TYPE DUT_DataRequest :
STRUCT
	aByte	: ARRAY[0..1] OF stByteAsBit; 	
	aDWord	: DWORD;
END_STRUCT
END_TYPE

(* stored: Version 1.1.0.1, ProductVersion 3.1.4024.15
   DUT DUT_DataRequest: Id {e6ebe229-be87-4cec-9bc0-990d3aaa44a0} *)
